# B&R Automation Studio project AGV (part 2)

#### ros_topics_typ.c - ros_topics_typ library source
```c
#include <ros_topics.h>

#define EXOS_ASSERT_LOG &handle->logger
#define EXOS_ASSERT_CALLBACK inst->_state = 255;
#include "exos_log.h"
#include "exos_ros_topics_typ.h"
#include <string.h>

#define SUCCESS(_format_, ...) exos_log_success(&handle->logger, EXOS_LOG_TYPE_USER, _format_, ##__VA_ARGS__);
#define INFO(_format_, ...) exos_log_info(&handle->logger, EXOS_LOG_TYPE_USER, _format_, ##__VA_ARGS__);
#define VERBOSE(_format_, ...) exos_log_debug(&handle->logger, EXOS_LOG_TYPE_USER + EXOS_LOG_TYPE_VERBOSE, _format_, ##__VA_ARGS__);
#define ERROR(_format_, ...) exos_log_error(&handle->logger, _format_, ##__VA_ARGS__);

int test;
int test2;

typedef struct
{
    void *self;
    exos_log_handle_t logger;
    ros_topics_typ data;

    exos_datamodel_handle_t ros_topics_typ_datamodel;

    exos_dataset_handle_t odemetry_dataset;
    exos_dataset_handle_t twist_dataset;
    exos_dataset_handle_t config_dataset;
    exos_dataset_handle_t encoder_dataset;
    exos_dataset_handle_t vaccumtopic;
    exos_dataset_handle_t linefollow;
    exos_dataset_handle_t linestatus;
} ros_topics_typHandle_t;

static void datasetEvent(exos_dataset_handle_t *dataset, EXOS_DATASET_EVENT_TYPE event_type, void *info)
{
    struct ros_topics_typCyclic *inst = (struct ros_topics_typCyclic *)dataset->datamodel->user_context;
    ros_topics_typHandle_t *handle = (ros_topics_typHandle_t *)inst->Handle;

    switch (event_type)
    {
    case EXOS_DATASET_EVENT_UPDATED:
        VERBOSE("dataset %s updated! latency (us):%i", dataset->name, (exos_datamodel_get_nettime(dataset->datamodel) - dataset->nettime));
        //handle each subscription dataset separately
        if(0 == strcmp(dataset->name, "twist"))
        {
            memcpy(&inst->pros_topics_typ->twist, dataset->data, dataset->size);
        }
        else if(0 == strcmp(dataset->name, "config"))
        {
            memcpy(&inst->pros_topics_typ->config, dataset->data, dataset->size);
        }
        else if(0 == strcmp(dataset->name, "vaccumTopic"))
        {
            memcpy(&inst->pros_topics_typ->vaccumTopic, dataset->data, dataset->size);
        }
        else if(0 == strcmp(dataset->name, "lineFollow"))
        {
            memcpy(&inst->pros_topics_typ->lineFollow, dataset->data, dataset->size);
        }
        break;

    case EXOS_DATASET_EVENT_PUBLISHED:
        VERBOSE("dataset %s published to local server for distribution! send buffer free:%i", dataset->name, dataset->send_buffer.free);
        //handle each published dataset separately
        if(0 == strcmp(dataset->name, "odemetry"))
        {
            // ros_topic_odemety_typ *odemetry_dataset = (ros_topic_odemety_typ *)dataset->data;
        }
        else if(0 == strcmp(dataset->name, "encoder"))
        {
            // ros_encoder *encoder_dataset = (ros_encoder *)dataset->data;
        }
        else if(0 == strcmp(dataset->name, "lineStatus"))
        {
            // ros_lineStatus *linestatus = (ros_lineStatus *)dataset->data;
        }
        break;

    case EXOS_DATASET_EVENT_DELIVERED:
        VERBOSE("dataset %s delivered to remote server for distribution! send buffer free:%i", dataset->name, dataset->send_buffer.free);
        //handle each published dataset separately
        if(0 == strcmp(dataset->name, "odemetry"))
        {
            // ros_topic_odemety_typ *odemetry_dataset = (ros_topic_odemety_typ *)dataset->data;
        }
        else if(0 == strcmp(dataset->name, "encoder"))
        {
            // ros_encoder *encoder_dataset = (ros_encoder *)dataset->data;
        }
        else if(0 == strcmp(dataset->name, "lineStatus"))
        {
            // ros_lineStatus *linestatus = (ros_lineStatus *)dataset->data;
        }
        break;

    case EXOS_DATASET_EVENT_CONNECTION_CHANGED:
        INFO("dataset %s changed state to %s", dataset->name, exos_get_state_string(dataset->connection_state));

        switch (dataset->connection_state)
        {
        case EXOS_STATE_DISCONNECTED:
            break;
        case EXOS_STATE_CONNECTED:
            //call the dataset changed event to update the dataset when connected
            //datasetEvent(dataset,EXOS_DATASET_UPDATED,info);
            break;
        case EXOS_STATE_OPERATIONAL:
            break;
        case EXOS_STATE_ABORTED:
            ERROR("dataset %s error %d (%s) occured", dataset->name, dataset->error, exos_get_error_string(dataset->error));
            break;
        }
        break;
    }

}

static void datamodelEvent(exos_datamodel_handle_t *datamodel, const EXOS_DATAMODEL_EVENT_TYPE event_type, void *info)
{
    struct ros_topics_typCyclic *inst = (struct ros_topics_typCyclic *)datamodel->user_context;
    ros_topics_typHandle_t *handle = (ros_topics_typHandle_t *)inst->Handle;

    switch (event_type)
    {
    case EXOS_DATAMODEL_EVENT_CONNECTION_CHANGED:
        INFO("application changed state to %s", exos_get_state_string(datamodel->connection_state));

        inst->Disconnected = 0;
        inst->Connected = 0;
        inst->Operational = 0;
        inst->Aborted = 0;

        switch (datamodel->connection_state)
        {
        case EXOS_STATE_DISCONNECTED:
            inst->Disconnected = 1;
            inst->_state = 255;
            break;
        case EXOS_STATE_CONNECTED:
            inst->Connected = 1;
            break;
        case EXOS_STATE_OPERATIONAL:
            SUCCESS("ros_topics_typ operational!");
            inst->Operational = 1;
            break;
        case EXOS_STATE_ABORTED:
            ERROR("application error %d (%s) occured", datamodel->error, exos_get_error_string(datamodel->error));
            inst->_state = 255;
            inst->Aborted = 1;
            break;
        }
        break;
    case EXOS_DATAMODEL_EVENT_SYNC_STATE_CHANGED:
        break;

    default:
        break;

    }

}

_BUR_PUBLIC void ros_topics_typInit(struct ros_topics_typInit *inst)
{
    ros_topics_typHandle_t *handle;
    TMP_alloc(sizeof(ros_topics_typHandle_t), (void **)&handle);
    if (NULL == handle)
    {
        inst->Handle = 0;
        return;
    }

    memset(&handle->data, 0, sizeof(handle->data));
    handle->self = handle;

    exos_log_init(&handle->logger, "gros_topics_typ_0");

    exos_datamodel_handle_t *ros_topics_typ_datamodel = &handle->ros_topics_typ_datamodel;
    exos_dataset_handle_t *odemetry_dataset = &handle->odemetry_dataset;
    exos_dataset_handle_t *twist_dataset = &handle->twist_dataset;
    exos_dataset_handle_t *config_dataset = &handle->config_dataset;
    exos_dataset_handle_t *encoder_dataset = &handle->encoder_dataset;
    exos_dataset_handle_t *vaccumtopic = &handle->vaccumtopic;
    exos_dataset_handle_t *linefollow = &handle->linefollow;
    exos_dataset_handle_t *linestatus = &handle->linestatus;
    EXOS_ASSERT_OK(exos_datamodel_init(ros_topics_typ_datamodel, "ros_topics_typ_0", "gros_topics_typ_0"));

    EXOS_ASSERT_OK(exos_dataset_init(odemetry_dataset, ros_topics_typ_datamodel, "odemetry", &handle->data.odemetry, sizeof(handle->data.odemetry)));
    EXOS_ASSERT_OK(exos_dataset_init(twist_dataset, ros_topics_typ_datamodel, "twist", &handle->data.twist, sizeof(handle->data.twist)));
    EXOS_ASSERT_OK(exos_dataset_init(config_dataset, ros_topics_typ_datamodel, "config", &handle->data.config, sizeof(handle->data.config)));
    EXOS_ASSERT_OK(exos_dataset_init(encoder_dataset, ros_topics_typ_datamodel, "encoder", &handle->data.encoder, sizeof(handle->data.encoder)));
    EXOS_ASSERT_OK(exos_dataset_init(vaccumtopic, ros_topics_typ_datamodel, "vaccumTopic", &handle->data.vaccumTopic, sizeof(handle->data.vaccumTopic)));
    EXOS_ASSERT_OK(exos_dataset_init(linefollow, ros_topics_typ_datamodel, "lineFollow", &handle->data.lineFollow, sizeof(handle->data.lineFollow)));
    EXOS_ASSERT_OK(exos_dataset_init(linestatus, ros_topics_typ_datamodel, "lineStatus", &handle->data.lineStatus, sizeof(handle->data.lineStatus)));

    inst->Handle = (UDINT)handle;
}

_BUR_PUBLIC void ros_topics_typCyclic(struct ros_topics_typCyclic *inst)
{
    ros_topics_typHandle_t *handle = (ros_topics_typHandle_t *)inst->Handle;

    inst->Error = false;
    if (NULL == handle || NULL == inst->pros_topics_typ)
    {
        inst->Error = true;
        return;
    }
    if ((void *)handle != handle->self)
    {
        inst->Error = true;
        return;
    }

    ros_topics_typ *data = &handle->data;
    exos_datamodel_handle_t *ros_topics_typ_datamodel = &handle->ros_topics_typ_datamodel;
    //the user context of the datamodel points to the ros_topics_typCyclic instance
    ros_topics_typ_datamodel->user_context = inst; //set it cyclically in case the program using the FUB is retransferred
    ros_topics_typ_datamodel->user_tag = 0; //user defined
    //handle online download of the library
    if(NULL != ros_topics_typ_datamodel->datamodel_event_callback && ros_topics_typ_datamodel->datamodel_event_callback != datamodelEvent)
    {
        ros_topics_typ_datamodel->datamodel_event_callback = datamodelEvent;
        exos_log_delete(&handle->logger);
        exos_log_init(&handle->logger, "gros_topics_typ_0");
    }

    exos_dataset_handle_t *odemetry_dataset = &handle->odemetry_dataset;
    odemetry_dataset->user_context = NULL; //user defined
    odemetry_dataset->user_tag = 0; //user defined
    //handle online download of the library
    if(NULL != odemetry_dataset->dataset_event_callback && odemetry_dataset->dataset_event_callback != datasetEvent)
    {
        odemetry_dataset->dataset_event_callback = datasetEvent;
    }

    exos_dataset_handle_t *twist_dataset = &handle->twist_dataset;
    twist_dataset->user_context = NULL; //user defined
    twist_dataset->user_tag = 0; //user defined
    //handle online download of the library
    if(NULL != twist_dataset->dataset_event_callback && twist_dataset->dataset_event_callback != datasetEvent)
    {
        twist_dataset->dataset_event_callback = datasetEvent;
    }

    exos_dataset_handle_t *config_dataset = &handle->config_dataset;
    config_dataset->user_context = NULL; //user defined
    config_dataset->user_tag = 0; //user defined
    //handle online download of the library
    if(NULL != config_dataset->dataset_event_callback && config_dataset->dataset_event_callback != datasetEvent)
    {
        config_dataset->dataset_event_callback = datasetEvent;
    }

    exos_dataset_handle_t *encoder_dataset = &handle->encoder_dataset;
    encoder_dataset->user_context = NULL; //user defined
    encoder_dataset->user_tag = 0; //user defined
    //handle online download of the library
    if(NULL != encoder_dataset->dataset_event_callback && encoder_dataset->dataset_event_callback != datasetEvent)
    {
        encoder_dataset->dataset_event_callback = datasetEvent;
    }

    exos_dataset_handle_t *vaccumtopic = &handle->vaccumtopic;
    vaccumtopic->user_context = NULL; //user defined
    vaccumtopic->user_tag = 0; //user defined
    //handle online download of the library
    if(NULL != vaccumtopic->dataset_event_callback && vaccumtopic->dataset_event_callback != datasetEvent)
    {
        vaccumtopic->dataset_event_callback = datasetEvent;
    }

    exos_dataset_handle_t *linefollow = &handle->linefollow;
    linefollow->user_context = NULL; //user defined
    linefollow->user_tag = 0; //user defined
    //handle online download of the library
    if(NULL != linefollow->dataset_event_callback && linefollow->dataset_event_callback != datasetEvent)
    {
        linefollow->dataset_event_callback = datasetEvent;
    }

    exos_dataset_handle_t *linestatus = &handle->linestatus;
    linestatus->user_context = NULL; //user defined
    linestatus->user_tag = 0; //user defined
    //handle online download of the library
    if(NULL != linestatus->dataset_event_callback && linestatus->dataset_event_callback != datasetEvent)
    {
        linestatus->dataset_event_callback = datasetEvent;
    }

    //unregister on disable
    if (inst->_state && !inst->Enable)
    {
        inst->_state = 255;
    }

    switch (inst->_state)
    {
    case 0:
        inst->Disconnected = 1;
        inst->Connected = 0;
        inst->Operational = 0;
        inst->Aborted = 0;

        if (inst->Enable)
        {
            inst->_state = 10;
        }
        break;

    case 10:
        inst->_state = 100;

        SUCCESS("starting ros_topics_typ application..");

        //connect the datamodel, then the datasets
        EXOS_ASSERT_OK(exos_datamodel_connect_ros_topics_typ(ros_topics_typ_datamodel, datamodelEvent));
        EXOS_ASSERT_OK(exos_dataset_connect(odemetry_dataset, EXOS_DATASET_PUBLISH, datasetEvent));
        EXOS_ASSERT_OK(exos_dataset_connect(twist_dataset, EXOS_DATASET_SUBSCRIBE, datasetEvent));
        EXOS_ASSERT_OK(exos_dataset_connect(config_dataset, EXOS_DATASET_SUBSCRIBE, datasetEvent));
        EXOS_ASSERT_OK(exos_dataset_connect(encoder_dataset, EXOS_DATASET_PUBLISH, datasetEvent));
        EXOS_ASSERT_OK(exos_dataset_connect(vaccumtopic, EXOS_DATASET_SUBSCRIBE, datasetEvent));
        EXOS_ASSERT_OK(exos_dataset_connect(linefollow, EXOS_DATASET_SUBSCRIBE, datasetEvent));
        EXOS_ASSERT_OK(exos_dataset_connect(linestatus, EXOS_DATASET_PUBLISH, datasetEvent));

        inst->Active = true;
        break;

    case 100:
    case 101:
        if (inst->Start)
        {
            if (inst->_state == 100)
            {
                EXOS_ASSERT_OK(exos_datamodel_set_operational(ros_topics_typ_datamodel));
                inst->_state = 101;
            }
        }
        else
        {
            inst->_state = 100;
        }

        EXOS_ASSERT_OK(exos_datamodel_process(ros_topics_typ_datamodel));
        //put your cyclic code here!

         if (exos_datamodel_get_nettime(odemetry_dataset->datamodel)- test > 28500 || exos_datamodel_get_nettime(odemetry_dataset->datamodel)- test < -28500  )
        {

            test = exos_datamodel_get_nettime(odemetry_dataset->datamodel);
            memcpy(&data->odemetry, &inst->pros_topics_typ->odemetry, sizeof(data->odemetry));
            exos_dataset_publish(odemetry_dataset);

        }

        if (exos_datamodel_get_nettime(odemetry_dataset->datamodel)- test2 > 1000000 || exos_datamodel_get_nettime(odemetry_dataset->datamodel)- test2 < -1000000  )
        {

            test2 = exos_datamodel_get_nettime(odemetry_dataset->datamodel);

            if (0 != memcmp(&inst->pros_topics_typ->lineStatus, &data->lineStatus, sizeof(data->lineStatus)))
            {
            memcpy(&data->lineStatus, &inst->pros_topics_typ->lineStatus, sizeof(data->lineStatus));
            exos_dataset_publish(linestatus);
            }

        }

        //}
        //}

        //publish the encoder_dataset dataset as soon as there are changes

        if (0 != memcmp(&inst->pros_topics_typ->encoder, &data->encoder, sizeof(data->encoder)))
        {
            memcpy(&data->encoder, &inst->pros_topics_typ->encoder, sizeof(data->encoder));
            exos_dataset_publish(encoder_dataset);
        }
        //publish the linestatus dataset as soon as there are changes

        break;

    case 255:
        //disconnect the datamodel
        EXOS_ASSERT_OK(exos_datamodel_disconnect(ros_topics_typ_datamodel));

        inst->Active = false;
        inst->_state = 254;
        //no break

    case 254:
        if (!inst->Enable)
            inst->_state = 0;
        break;
    }

    exos_log_process(&handle->logger);

}

_BUR_PUBLIC void ros_topics_typExit(struct ros_topics_typExit *inst)
{
    ros_topics_typHandle_t *handle = (ros_topics_typHandle_t *)inst->Handle;

    if (NULL == handle)
    {
        ERROR("ros_topics_typExit: NULL handle, cannot delete resources");
        return;
    }
    if ((void *)handle != handle->self)
    {
        ERROR("ros_topics_typExit: invalid handle, cannot delete resources");
        return;
    }

    exos_datamodel_handle_t *ros_topics_typ_datamodel = &handle->ros_topics_typ_datamodel;

    EXOS_ASSERT_OK(exos_datamodel_delete(ros_topics_typ_datamodel));

    //finish with deleting the log
    exos_log_delete(&handle->logger);
    //free the allocated handle
    TMP_free(sizeof(ros_topics_typHandle_t), (void *)handle);
}
```

### VisionTypes.typ
```iecst
(*-----------------------------------------------------------------------------------------------------------------------------------------*)
(*General vision structures*)

TYPE
	typVisionMain : 	STRUCT
		CMD : typVisionCommand;
		CFG : typVisionConfig;
		DAT : typVisionData;
		FCT : typVisionFunction;
		DIA : typVisionDiag;
		OPT : typVisionOptics;
		HW : typVisionHW;
	END_STRUCT;
	typVisionCommand : 	STRUCT
		ImageTrigger : BOOL;
		ImageTriggerReset : BOOL;
		AutoSetupStartStop : BOOL;
		VaSwitchApplication : BOOL;
		SaveDiagData : BOOL;
		ReadCameraInfo : BOOL;
	END_STRUCT;
	typVisionConfig : 	STRUCT
		VisionFunction : enumVisionFunction;
		PowerlinkNode : USINT;
		DataStructure : UDINT;
		ComponentLink : ViComponentType;
		ResolutionWidth_X : UINT; (*Nr of sensor pixels in x direction (width). Is always bigger than height*)
		ResolutionHeight_Y : UINT; (*Nr of sensor pixels in y direction (height). Is always smaller than width*)
	END_STRUCT;
	typVisionFunction : 	STRUCT
		ApplicationName : STRING[40];
		Status : DINT;
	END_STRUCT;
	typVisionDiag : 	STRUCT
		DiagName : STRING[80] := 'diag.tgz';
		Status : DINT;
	END_STRUCT;
	typVisionData : 	STRUCT
		Enable : BOOL := FALSE;
		MaxItemCnt : USINT := 10;
		NettimeDelay : DINT;
		Timeout : UINT := 5000;
		Gain : USINT;
		Focus : UINT;
		Exposure : UDINT;
		FlashColor : USINT := 1;
		FlashSegment : USINT := 15;
		LedColor : USINT;
		IRFilter : BOOL;
		OffsetROIX : DINT;
		OffsetROIY : DINT;
		OffsetROIRotationCenterX : DINT;
		OffsetROIRotationCenterY : DINT;
		OffsetROIOrientation : INT;
		ChromaticLock : BOOL;
		Alignment : USINT;
		AutoSetupGain : USINT;
		AutoSetupFocus : UINT;
		AutoSetupExposure : UDINT;
		AcquisitionAcceptedCnt : USINT;
		AcquisitionCompletedCnt : USINT;
		AcquisitionFailedCnt : USINT;
		LightWarningCnt : USINT;
		ImageProcessingError : UINT;
		ImageProcessingActive : BOOL;
		ImageNettime : DINT;
		ProcessingTimeCamera : UINT;
		ProcessingTimeFunction : UINT;
		ResultCnt : USINT;
		CockpitIsActive : BOOL;
		Status : UDINT;
		StatusText : STRING[30];
		Active : BOOL;
	END_STRUCT;
	typVisionOptics : 	STRUCT
		OrderNr : STRING[40];
		Binning : BOOL;
		ResolutionX : INT;
		ResolutionY : INT;
		Lens : USINT;
		Sensor : USINT;
		ValidDistance : BOOL;
		Distance_mm : LREAL;
		DistanceLens_mm : LREAL;
		HyperFocalDistance_mm : LREAL;
		PixelSize_um : LREAL;
		PixelSizeBinning_um : LREAL;
		FocalLength_mm : LREAL;
		MinObjectDist_mm : LREAL;
		MaxObjectDist_mm : LREAL;
		Aperture : LREAL;
		CircleOfConfusion_mm : LREAL;
		DepthOfFieldNearPos_mm : LREAL;
		DepthOfFieldFarPos_mm : LREAL;
		DepthOfField_mm : LREAL;
		FieldOfView_X_mm : LREAL;
		FieldOfView_Y_mm : LREAL;
		Resolution_mmPerPx : LREAL;
	END_STRUCT;
	typVisionHW : 	STRUCT
		Connected : BOOL;
		Ready : BOOL;
		DigitalInput01 : BOOL;
		DigitalOutput01 : BOOL;
		DigitalOutputStatus01 : BOOL;
		DigitalOutput02 : BOOL;
		DigitalOutputStatus02 : BOOL;
		SerialNumber : UDINT;
		ID : UDINT;
		Variant : UDINT;
		Firmware : UDINT;
		Undervoltage : BOOL;
		Temperature : SINT;
	END_STRUCT;
	enumVisionFunction :
		(
		enumFunctionNone,
		enumBlob
		);
END_TYPE

(*-----------------------------------------------------------------------------------------------------------------------------------------*)
(*General Light structures*)
(*-----------------------------------------------------------------------------------------------------------------------------------------*)
(*General nettime structures*)

TYPE
	typVisionNettime : 	STRUCT
		CMD : typNettimeCommand;
		CFG : typNettimeConfig;
		DAT : typNettimeData;
	END_STRUCT;
	typNettimeCommand : 	STRUCT
		Activate : BOOL;
	END_STRUCT;
	typNettimeConfig : 	STRUCT
		AxisPeriod : LREAL; (*Units when period repeats*)
		AxisPositionTrigger : LREAL; (*Position in the period where trigger is fired*)
		AxisPositionDelay_Cycles : LREAL; (*Delay in PLK cycles for the read position from drive*)
		VisionPreTrigger_Cycles : DINT; (*Number of powerlink cycles the trigger has to be send ahead*)
	END_STRUCT;
	typNettimeData : 	STRUCT
		NettimeNext_us : DINT; (*Calculated nettime for next trigger*)
		NettimeDelta_us : DINT; (*Difference between current nettime and calculated nettime for the camera trigger*)
		AxisPosition : LREAL; (*Current axis position*)
		AxisVelocity : LREAL; (*Current axis position*)
		AxisInVelocity : BOOL; (*Indicates that the axis is moving at speed*)
		Overflow : DINT; (*Counts up when a trigger could not be set on time*)
	END_STRUCT;
END_TYPE

(*-----------------------------------------------------------------------------------------------------------------------------------------*)
(*Color detection structures*)

TYPE
	typVisionColor : 	STRUCT
		CMD : typVisionColorCommand;
		CFG : typVisionColorConfig;
		DAT : typVisionColorData;
	END_STRUCT;
	typVisionColorCommand : 	STRUCT
		Evaluate : BOOL; (*Evaluate new product and try to determine the color*)
		Teach : BOOL; (*Teach a new product and store color information*)
		ResetError : BOOL; (*Reset error state*)
	END_STRUCT;
	typVisionColorConfig : 	STRUCT
		FlashColor1 : USINT := 1; (*First flash color (red)*)
		FlashColor2 : USINT := 2; (*Second flash color (green)*)
		FlashColor3 : USINT := 3; (*Third flash color (blue)*)
		FlashColor4 : USINT := 4; (*Fourth flash color (lime)*)
		ProductName : ARRAY[1..MAX_NUM_PRODUCTS]OF STRING[80]; (*Name of the product*)
		GrayValue1 : ARRAY[1..MAX_NUM_PRODUCTS]OF UINT; (*Mean gray value for first flash color*)
		GrayValue2 : ARRAY[1..MAX_NUM_PRODUCTS]OF UINT; (*Mean gray value for second flash color*)
		GrayValue3 : ARRAY[1..MAX_NUM_PRODUCTS]OF UINT; (*Mean gray value for third flash color*)
		GrayValue4 : ARRAY[1..MAX_NUM_PRODUCTS]OF UINT; (*Mean gray value for fourth flash color*)
		TeachingIndex : UINT(1..1000)  := 1; (*Index that is currently taught*)
		MaxError : UINT := 100; (*Maximum error for all gray values*)
		MinDifference : UINT := 10; (*Minimum distance to next best value*)
	END_STRUCT;
	typVisionColorData : 	STRUCT
		GrayValue1 : UINT; (*Current mean gray value for first flash color*)
		GrayValue2 : UINT; (*Current mean gray value for second flash color*)
		GrayValue3 : UINT; (*Current mean gray value for third flash color*)
		GrayValue4 : UINT; (*Current mean gray value for fourth flash color*)
		TotalError : ARRAY[1..MAX_NUM_PRODUCTS]OF UINT; (*Total error of mean gray value for all products*)
		LowError : UINT; (*Lowest error found*)
		LowDistance : UINT; (*Distance to next best value*)
		LowIndex : UINT; (*Index of the best value*)
		LowName : STRING[80]; (*Product name of the best value*)
		Status : UINT; (*Status of color detection*)
	END_STRUCT;
END_TYPE

(*-----------------------------------------------------------------------------------------------------------------------------------------*)
(*Image upload structures*)

TYPE
	typVisionImage : 	STRUCT
		CMD : typVisionImageCommand;
		CFG : typVisionImageConfig;
		DAT : typVisionImageData;
	END_STRUCT;
	typVisionImageCommand : 	STRUCT
		CreateDir : BOOL;
		DeleteDir : BOOL;
		DeleteImage : BOOL;
		Refresh : BOOL;
		DownloadImage : BOOL;
		SaveImageOnPLC : BOOL;
		ResetError : BOOL;
		RefreshCrosshair : BOOL;
	END_STRUCT;
	typVisionImageConfig : 	STRUCT
		FileDevice : STRING[80];
		DirName : STRING[80];
		PlkIPWithoutNode : STRING[80];
		EthDevice : STRING[80];
		EthIP : STRING[80];
		ConvertCycles : UDINT;
		Format : USINT; (*0: jpg. 1: bmp*)
		QualityJPG : USINT;
		UploadBmpJpg : BOOL;
		UploadSVG : BOOL;
		MainPageQualityJPG : USINT; (*quality of the jpg image on the main page. min:0, max:100, good value: 30*)
		ImageRotation_deg : UINT; (*rotation of the whole image, steps in degree. Only values 0, 90. 180, 270 make sense*)
	END_STRUCT;
	typVisionImageData : 	STRUCT
		Images : ARRAY[0..19]OF STRING[80];
		Status : UINT;
		VisionDisabled : BOOL;
	END_STRUCT;
END_TYPE

(*-----------------------------------------------------------------------------------------------------------------------------------------*)
(*Vision specific structures*)

TYPE
	typBlobMain : 	STRUCT  (*Blob function structures*)
		RegionalFeature : BOOL;
		EnhancedBlobInformation : BOOL := FALSE;
		ModelNumber : ARRAY[1..MAX_NUM_RESULTS]OF USINT;
		Clipped : ARRAY[1..MAX_NUM_RESULTS]OF BOOL;
		Area : ARRAY[1..MAX_NUM_RESULTS]OF UDINT;
		PositionX : ARRAY[1..MAX_NUM_RESULTS]OF DINT;
		PositionY : ARRAY[1..MAX_NUM_RESULTS]OF DINT;
		Orientation : ARRAY[1..MAX_NUM_RESULTS]OF INT;
		MeanGrayValue : ARRAY[1..MAX_NUM_RESULTS]OF USINT;
		Length : ARRAY[1..MAX_NUM_RESULTS]OF UDINT;
		Width : ARRAY[1..MAX_NUM_RESULTS]OF UDINT;
	END_STRUCT;
END_TYPE

(*------------------------------------------------------------------------------------------------------------------------------------------------------------------------------------------------------------------------*)
(*Structure that contains the recipe variables*)

TYPE
	recVariable : 	STRUCT
		Cam : ARRAY[1..MAX_NUM_CAMS]OF recVariableCam;
		Light : ARRAY[1..10]OF recVariableLight;
	END_STRUCT;
	recVariableCam : 	STRUCT
		ApplicationName : STRING[40];
		MaxItemCnt : USINT := 10;
		Timeout : UINT := 5000;
		Gain : USINT;
		Focus : UINT;
		Exposure : UDINT;
		FlashColor : USINT := 1;
		FlashSegment : USINT := 15;
	END_STRUCT;
	recVariableLight : 	STRUCT
		Timeout : UINT := 5000;
		Exposure : UDINT;
		FlashColor : USINT := 1;
		FlashSegment : UINT := 15;
		SetAngle : UINT := 45;
	END_STRUCT;
END_TYPE
```

### VisionVariables.var
```iecst
(*-----------------------------------------------------------------------------------------------------------------------------------------*)
(*Global variables for sensor hardware and vision functions*)
VAR
	gBlob : typBlobMain; (*Data that is specific for the blob function*)
	gVisionColor : typVisionColor;
	gVisionImage : typVisionImage; (*Data for image handling*)
	gVisionNettime : typVisionNettime; (*Data for nettime calculation*)
	gVisionSensor : ARRAY[0..MAX_NUM_CAMS] OF typVisionMain; (*General vision functions that are independent from the inspection function*)
	gSelectedSensor : UINT := 1; (*Selected camera node number*)
	NettimeCurrent_us : DINT; (*Current Powerlink nettime*)
END_VAR
VAR RETAIN
	Recipedata : recVariable;
END_VAR
(*
	RecipeData : recVariable; (*Structure that contains the recipe variables*)
(*-----------------------------------------------------------------------------------------------------------------------------------------*)
(*Global constants*)
VAR CONSTANT
	MAX_NUM_CAMS : UINT := 1; (*Maximum number of camera's*)
	MAX_NUM_LIGHTS : UINT := 10; (*Maximum number of light's*)
	MAX_NUM_RESULTS : UINT := 10; (*Maximum number of results*)
	MAX_NUM_PRODUCTS : UINT := 8; (*Maximum number of products for color detection*)
	MAX_IDX_VA_LIST : UINT := 19; (*Maximum number of entrys in the Vision Application list*)
	DEVICE_NAME : STRING[40] := 'VisionFileDevice'; (*File device where the images and recipes are stored*)
	NETTIME_DEFAULT_DELAY : UDINT := 30000; (*This delay is used when software trigger is used and nettime is enabled*)
	NETTIME_ENABLE : BOOL := FALSE; (*Enable nettime code, this generates the nettime when using manual triggers*)
	MAX_NUM_CODETYPES : USINT := 69; (*Maximum number of code types*)
END_VAR
VAR
	CodeTypes : {REDUND_UNREPLICABLE} ARRAY[0..MAX_NUM_CODETYPES] OF STRING[80] := ['Auto Identify (0)','2/5 Industrial (1)','2/5 Interleaved (2)','Codebar (3)','Code 32 (4)','Code 39 (5)','Code 93 (6)','Code 128 (7)','MSI (8)','PharmaCode (9)','EAN-8 (10)','EAN-8 Add-On 2 (11)','EAN-8 Add-On 5 (12)','EAN-13 (13)','EAN-13 Add-On 2 (14)','EAN-13 Add-On 5 (15)',4(''),'UPC-A (20)','UPC-A Add-On 2 (21)','UPC-A Add-On 5 (22)','UPC-E (23)','UPC-E Add-On 2 (24)','UPC-E Add-On 5 (25)',4(''),'GS1-128 (30)','GS1 DataBar Omnidirectional (31)','GS1 DataBar Truncated (32)','GS1 DataBar Stacked (33)','GS1 DataBar Stacked Omnidirectional (34)','GS1 DataBar Limited (35)','GS1 DataBar Expanded (36)','GS1 DataBar ExpandedStacked (37)',12(''),'Data Matrix ECC200 (50)','QR Code Model 1 (51)','QR Code Model 2 (52)','Micro QRCode (53)','PDF417 (54)','Aztec Code (55)',4(''),'GS1 Data Matrix (60)','GS1 QR Code Model 1 (61)','GS1 QR Code Model 2 (62)','GS1 Aztec Code (63)',6('')]; (*Codes types for code reading*)
END_VAR
```

### Program Logical/Package/VisionMain (IEC)

#### Cyclic1.st
```iecst
PROGRAM _CYCLIC

//	/// PARAMETER//////////////////////

	gVisionImage.CFG.EthDevice := 'IF2';
	gVisionSensor[0].CFG.VisionFunction := enumBlob;
	gVisionSensor[0].CFG.PowerlinkNode := 1;
	gVisionSensor[0].CFG.DataStructure := ADR(gBlob);
	gVisionSensor[0].CFG.ComponentLink := gCamera;
//
//
//

	hwBlob.out.common.enable := TRUE;
	hwBlob.out.common.numSearchMax := 10;
	hwBlob.out.enhancedBlobInformation := TRUE;
	hwBlob.out.regionFeatures := TRUE;
	hwBlob.out.common.alignment := 0;
	hwBlob.out.common.offsetROI.orientation := 0;
	hwBlob.out.common.offsetROI.rotCenterX := 0;
	hwBlob.out.common.offsetROI.rotCenterY := 0;
	hwBlob.out.common.offsetROI.x := 0;
	hwBlob.out.common.offsetROI.y := 0;
	hwCam.out.par.focus := 11000;
	hwCam.out.par.flashColor := 99;
	hwCam.out.par.flashSegment := 4;
	hwCam.out.par.exposureTime := 1000;
	imgTrig.pCameraHw := ADR(hwCam);

	//// PARAMETER///////////////////////////

IF hwCam.in.status.imageAcquisitionReady AND NOT hwCam.in.status.imageProcessingActive THEN
	imgTrig.trigger := TRUE;
		cnt := 0;

		// Vi starter med at kigge om vores kamera har fundet nogen resultater
		// Hvis der er resultater så begynder vi at proccess dem
		IF hwBlob.in.common.numResults <> 0 AND orientationReached AND NOT awaitDecision THEN

				// Først vil vi gerne gemme det index af vores resultater som er  vores linje
				// model 1 er den model der bruges til at finde linjen
				// det index som indeholder linjen bliver gemt i test
				// Ellers så tjekker vi om resultatet er fra den model som finder gulvet
			// indexet bliver gemt i et array af int's

			FOR i := 0 TO hwBlob.in.common.numResults BY 1 DO
				IF hwBlob.in.results[i].modelNumber = 1 THEN
					test := i;
				ELSIF hwBlob.in.results[i].modelNumber = 2 THEN
					floorIndex[cnt] := i;
					cnt := cnt+1;

				END_IF
			END_FOR
				// her tager vi de forskellige blob resultater af linjen som vi er intersseret i baseret på det index som vi gemte før
				minYPos := hwBlob.in.results[test].yMin/100;
				minXPos := hwBlob.in.results[test].xMin/100;
				maxYPos := hwBlob.in.results[test].yMax/100;
				maxXPos := hwBlob.in.results[test].xMax/100;
				posY := hwBlob.in.results[test].positionY/100;
				posX := hwBlob.in.results[test].positionX/100;
				middleY := (minYPos + maxYPos)/2;
				middleX := (minXPos + maxXPos)/2;
				xPosDiff := middleX-640;
				blobArea := hwBlob.in.results[test].area/100;

			// her resetter vi vores gulv index så vi ikke ved en fejl kommer til at tage et tidligere index fra sidste cycle
				prevFloorIndex := 10;
				// her går vi igennem alle de indexs som indeholder resultater fra gulvet
				// Bemærk at nogle index kan være 0 for alle resultater da det er baseret på hvor mange blobs kameraet finder
			FOR i := 0 TO 2 BY 1 DO
				IF floorIndex[i] <> prevFloorIndex THEN // muligvis ikke nødvendigt men bare for at være sikker så tjekker jeg at det ikke er det samme index vi gemmer flere gange
					floorBlob[i].maxXPos := hwBlob.in.results[floorIndex[i]].xMax/100;
					floorBlob[i].maxYPos := hwBlob.in.results[floorIndex[i]].yMax/100;
					floorBlob[i].minXPos := hwBlob.in.results[floorIndex[i]].xMin/100;
					floorBlob[i].minYPos := hwBlob.in.results[floorIndex[i]].yMin/100;
					floorBlob[i].circ := hwBlob.in.results[floorIndex[i]].circularity;
					floorBlob[i].area := hwBlob.in.results[floorIndex[i]].area/100;
					floorBlob[i].yPos := hwBlob.in.results[floorIndex[i]].positionY/100;
					floorBlob[i].rect := hwBlob.in.results[floorIndex[i]].rectangularity;
					floorBlob[i].xPos := hwBlob.in.results[floorIndex[i]].positionX;
					prevFloorIndex := floorIndex[i];
				END_IF

			END_FOR

				// logikken bag at finde om der er en 90 grader sving
				// essentielt så kigger den om vores gulv blob ligger imellem x og y-max + min af vores linje blob
				// tilføj illustration for dette
				// muligvis tilføj noget der tjekker hvor rektangulær gulv blobben er, hvis den ikke er rektangulær er det nok en sammenfletning istedet for
//			IF floorBlob[0].rect < 90 OR cnt < 1  THEN
//				conditionX := TRUE;
//				conditionY := TRUE;
//			ELSE
//				conditionX := floorBlob[0].minXPos+75 > maxXPos-75 OR floorBlob[0].maxXPos -75 < minXPos+75; //OR floorBlob[1].minXPos +50 > maxXPos-50 OR floorBlob[1].maxXPos -50 < minXPos+50;
//
//				conditionY := floorBlob[0].maxYPos -75 > minYPos +75 OR floorBlob[0].minYPos +75 < maxYPos-75; //OR floorBlob[1].maxYPos -50 > minYPos +50 OR floorBlob[1].minYPos +50 < maxYPos-50;
//
//			END_IF
//
//			conditionCheck := conditionX AND conditionY;
//
//			IF NOT conditionCheck THEN
//				awaitDecision := TRUE;
//			END_IF
//
//

				// Her tjekker vi om linjen bliver størrer, dette dækker tilfældet af sammenfletninger
			IF blobArea > 800000 THEN

				crossBool := TRUE;
				IF crossBool <> prevCrossBool THEN
					awaitDecision := TRUE;
					updateLineStatus := TRUE;
				END_IF

				prevCrossBool := crossBool;
			ELSE
				crossBool := FALSE;
				prevCrossBool := crossBool;
			END_IF

				// Hvis det er tilfældet af en sammenfletning så baseret på vores condition "holdRight" så drejer robotten til højre eller venstre
				// dette burde at lede robotten til en af de linjer der sammenflettes
				// derefter vil den gå tilbage til sit sædvanelige program
			IF crossBool AND (lineFollow.lineInterSection OR sammenEnable) THEN
				IF lineFollow.lineHoldRight OR holdRight THEN
					angle := 0.60;
				ELSE
					angle := -0.60;
	//				angle := -1.5707;
				END_IF
				// her udregner vi vinklen i mellem midten af kameraet og centeret af linje bloben
				// vi antager at det er en retvinklet trekant
					// tilføj illustration

					// i tilfældet af linjen er lige på så er vinkel super lille og dermed bliver differencen mellem vores hjul minimal
					// ellers så bliver forskellen i hastigheden i mellem hjullene størrer baseret på vinklen
					// essentielt så virker det som en simpel P-controller
				// kunne udvides med et D komponentet til at håndtere noget overshoot på justeringen

			ELSE

				angle := ASIN((640-posX)/SQRT(EXPT((640-posX),2)+EXPT((posY),2)));
			END_IF
			conditionCheck := minYPos < 10 AND maxYPos < 800;
			IF conditionCheck AND NOT crossBool THEN
				//awaitDecision := TRUE;
			END_IF
			// her bestemmes den mode som giver værdier til motoren
//				IF NOT conditionCheck AND (lineFollow.lineSharpTurn OR sharpTurn) THEN
//					updateLineStatus := TRUE;
//
//				IF floorBlob[0].yPos > 512 AND floorBlob[0].xPos > 640 THEN
//					angle := 0.01;
//					drejMere := angle;
//					rightTurn := FALSE;
//				ELSIF floorBlob[0].yPos < 512 AND floorBlob[0].xPos < 640 THEN
//					rightTurn := TRUE;
//					angle := -0.01;
//					drejMere := angle;
//				END_IF
//				orientationReached := FALSE;
//				Test2 := 20;			// som kan ses så hvor meget vi drejer er baseret på vinklen
				// vores reference angle vil være 0 i dette tilfælde da det vil være samme orientation som linjen
			IF crossBool AND (lineFollow.lineInterSection OR sammenEnable) THEN
				Test2 := 2;
				drejMere := angle;
				sammenEnable := FALSE;
			ELSIF sharpTurn THEN
				iVisionAlive := iVisionAlive +1;
				Test2 := 20;
				angle := -0.01;
				drejMere := angle;
			ELSIF maxYPos < 1023 AND minYPos > 10 AND (moveForward OR lineFollow.lineForward) THEN
				angle := 0.01;
				Test2 := -1;
				drejMere := angle;

			ELSIF (xPosDiff > 0 OR xPosDiff < 0) AND orientationReached THEN //venstre
				Test2 := 1;
				drejMere := angle;

//			ELSIF orientationReached THEN
//				Test2 := 10;
//				IF angle < 0 THEN
//					drejMere := -0.16;
//				ELSE
//					drejMere := 0.16;
//				END_IF
			END_IF
//
		ELSIF awaitDecision THEN
			Test2 := 0;
		ELSIF orientationReached THEN

		Test2 := 5;
		IF angle < 0 THEN
			drejMere := -0.16;
		ELSE
			drejMere := 0.16;
		END_IF
			// i tilfældet af at  vi ikke finder nogen resultater med kameraet så vil robotten rotere til den retning den sidste ville til
			// dette er for at at lave noget recovery i tilfælde af robotten mister linjen
			// den kunne ende med at rotere helt om sig selv og dermed finde linjen tilbage

	END_IF
		//		END_IF

END_IF

	imgTrig();

END_PROGRAM
```

#### Init1.st
```iecst
PROGRAM _INIT

	gVisionNettime.CMD.Activate := TRUE;
	gVisionNettime.CFG.AxisPeriod := 360;
	gVisionNettime.CFG.AxisPositionDelay_Cycles := 1;
	gVisionNettime.CFG.VisionPreTrigger_Cycles:= 8;

END_PROGRAM
```

#### Types.typ - Local data types
```iecst
TYPE
	blobPositions : 	STRUCT
		maxXPos : REAL;
		minXPos : REAL;
		maxYPos : REAL;
		minYPos : REAL;
		middleX : REAL;
		middleY : REAL;
		area : REAL;
		angle : REAL;
		rect : USINT;
		circ : USINT;
		yPos : REAL;
		xPos : REAL;
	END_STRUCT;
END_TYPE
```

#### Variables.var
```iecst
VAR
	angle : REAL;
	blobArea : UDINT;
	cnt : USINT;
	conditionCheck : BOOL;
	conditionX : BOOL;
	conditionY : BOOL;
	crossBool : BOOL;
	floorBlob : ARRAY[0..2] OF blobPositions;
	floorIndex : ARRAY[0..2] OF USINT;
	hwBlob : brdkViBase_hw_blob_10_typ;
	hwBlobFloor : brdkViBase_hw_blob_1_typ;
	hwCam : brdkViBase_cam_hw_typ;
	i : USINT;
	imgTrig : brdkViBase_imgTrigger;
	iVisionAlive : USINT;
	maxXPos : REAL;
	maxYPos : REAL;
	middleErr : REAL;
	middleX : REAL;
	middleY : REAL;
	minXPos : REAL;
	minYPos : REAL;
	posX : REAL;
	posY : REAL;
	prevCrossBool : BOOL;
	prevFloorIndex : USINT;
	sammenEnable : BOOL;
	test : INT;
	updateStatus : BOOL;
	xPosDiff : REAL;
END_VAR
```

#### evaluateStatus.st - not listed in the package file held
```iecst
ACTION evaluateStatus:

	IF lineFollow.lineMode THEN
		lineStatus.lineStatusCode := lineStatus.lineStatusCode +1;
	END_IF
	IF lineFollow.lineSharpTurn THEN
		lineStatus.lineStatusCode := lineStatus.lineStatusCode + 12;
	END_IF
	IF lineFollow.lineForward THEN
		lineStatus.lineStatusCode := lineStatus.lineStatusCode + 10;
	END_IF
	IF lineFollow.lineHoldRight THEN
		lineStatus.lineStatusCode := lineStatus.lineStatusCode + 2;
	END_IF
	IF lineFollow.lineInterSection THEN
		lineStatus.lineStatusCode := lineStatus.lineStatusCode + 14;
	END_IF

	updateLineStatus := TRUE;

END_ACTION
```

Listed in the project but not available here: Logical/Global.typ, Logical/ros_topics_typ/Linux/exos_ros_topics_typ.c, Logical/ros_topics_typ/motorCtrl/setupPointers.st, Logical/ros_topics_typ/motorCtrl/evaluateStatus.st, Logical/ros_topics_typ/ros_topics/exos_ros_topics_typ.h, Logical/ros_topics_typ/ros_topics/ros_topics.fun, Logical/ros_topics_typ/ros_topics/heapsize.cpp
